SUBAPPLICATION Uebung_012c (* Numeric Value Input und Speichern *)
  (* Standard: 61499-2 *)
  (* Version 1.0, 2023-10-23, franz *)
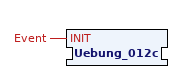
  EVENT_INPUT
    INIT;
  END_EVENT
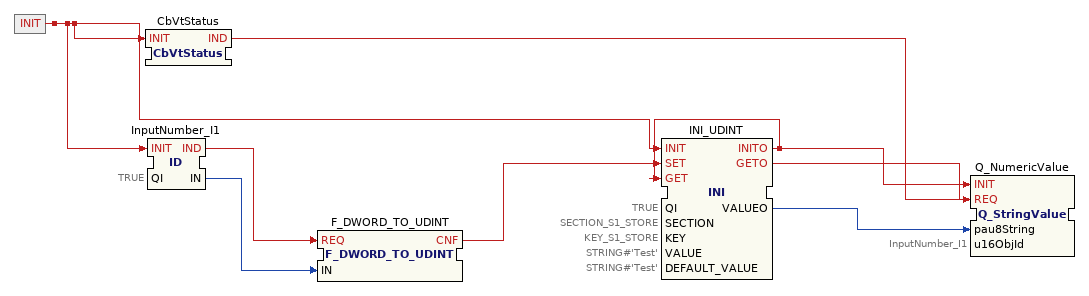
  FBS
    F_DWORD_TO_UDINT : F_DWORD_TO_UDINT;
    InputNumber_I1 : ID(QI := TRUE);
    INI_UDINT : INI(QI := TRUE, SECTION := SECTION_S1_STORE, KEY := KEY_S1_STORE, VALUE := STRING#'Test', DEFAULT_VALUE := STRING#'Test');
    Q_NumericValue : Q_StringValue(u16ObjId := InputNumber_I1);
    CbVtStatus : CbVtStatus;
  END_FBS
  EVENT_CONNECTIONS
    InputNumber_I1.IND TO F_DWORD_TO_UDINT.REQ;
    INIT TO InputNumber_I1.INIT;
    INIT TO CbVtStatus.INIT;
    INIT TO INI_UDINT.INIT;
    F_DWORD_TO_UDINT.CNF TO INI_UDINT.SET;
    INI_UDINT.INITO TO INI_UDINT.GET;
    INI_UDINT.INITO TO Q_NumericValue.INIT;
    CbVtStatus.IND TO Q_NumericValue.REQ;
    INI_UDINT.GETO TO Q_NumericValue.REQ;
  END_CONNECTIONS
  DATA_CONNECTIONS
    InputNumber_I1.IN TO F_DWORD_TO_UDINT.IN;
    INI_UDINT.VALUEO TO Q_NumericValue.pau8String;
  END_CONNECTIONS
END_SUBAPPLICATION
